	IF ((garPositionEndProcCalc[1] - T_Station_Parameter.T_StProcess.rPositionStartProc) <> 0.0) AND (T_Station_Parameter.T_OnlineChange.rWorkingSpeedForward <> 0.0) THEN
		T_Station_Work.THWWorkStation.TCtrlWork.iProgressBar_ZPos:=		REAL_TO_INT(100.0/(garPositionEndProcCalc[1] - T_Station_Parameter.T_StProcess.rPositionStartProc)
																			*(ptrTAxisZ^.T_LiveValue.lrActualPosition - T_Station_Parameter.T_StProcess.rPositionStartProc));
		T_Station_Work.THWWorkStation.TCtrlWork.iProgressBar_ZVel:=	REAL_TO_INT((100.0/T_Station_Parameter.T_OnlineChange.rWorkingSpeedForward)*ptrTAxisZ^.T_LiveValue.lrActualVelocity);
	ELSE
		T_Station_Work.THWWorkStation.TCtrlWork.iProgressBar_ZPos:=	0;
		T_Station_Work.THWWorkStation.TCtrlWork.iProgressBar_ZVel:=	0;
	END_IF;
	IF (T_Station_Work.THWWorkStation.TCtrlWork.iProgressBar_ZPos < 0) THEN
		T_Station_Work.THWWorkStation.TCtrlWork.iProgressBar_ZPos:=0;
	END_IF;
	IF (T_Station_Work.THWWorkStation.TCtrlWork.iProgressBar_ZVel < 0) THEN
		T_Station_Work.THWWorkStation.TCtrlWork.iProgressBar_ZVel:=0;
	END_IF;
(***************************************************************************************************************************************************)
(* Drehmoment Min-Max Werte oberhalb eines HC *)
rActTorque:=T_Station_Work.THWWorkStation.TCtrlWork.iProgressBar_Torque;
IF xStartFunction AND (iStationFunctionNr = 5) THEN
	IF (iStFct_StepPrc = 3) OR (iStFct_StepPrc = 4) THEN
		IF (rActTorque >= rTorqueMax) THEN
			rTorqueMax:=rActTorque;
		END_IF;
		IF (rActTorque >= rTorqueMin) THEN
			rTorqueMin:=rActTorque;
		END_IF;
	ELSE
		IF (T_Station_Work.THWWorkStation.TCtrlWork.iOverLimitCounterTorque >= 1) THEN
			IF (rTorqueMin <= rTorqueMin_Min) AND (rTorqueMin <> 0.0) AND (rTorqueMin >= 100.0)THEN
				rTorqueMin_Min:=rTorqueMin;
			END_IF;
			rTorqueMin:=0.0;
			IF (rTorqueMin_Min <> 99999.0) THEN
				T_Station_Work.THWWorkStation.TCtrlWork.rTorqueAfterHC_Min:=rTorqueMin_Min;
			END_IF;
		END_IF;
	END_IF;
	IF (rTorqueMax >= rTorqueMax_Max) THEN
		rTorqueMax_Max:=rTorqueMax;
	END_IF;
	T_Station_Work.THWWorkStation.TCtrlWork.rTorqueAfterHC_Max:=rTorqueMax_Max;
	IF (T_Station_Work.THWWorkStation.TCtrlWork.rTorqueAfterHC_Min <> 0.0) AND (T_Station_Work.THWWorkStation.TCtrlWork.rTorqueAfterHC_Min < 100.0) THEN
		T_Station_Work.THWWorkStation.TCtrlWork.rTorqueAfterHC_Min:=100.0;
	END_IF;
ELSE
	rTorqueMin:=0;
	rTorqueMax:=rActTorque;
	rTorqueMax_Max:=0;
	rTorqueMin_Min:=99999.0;
END_IF;
IF (T_Station_Work.THWWorkStation.TCtrlWork.rTorqueAfterHC_Min >= T_Station_Parameter.T_StProcess.iMaxTorque) THEN
	T_Station_Work.THWWorkStation.TCtrlWork.xTorqueAfterHC_Min_Overlimit:=TRUE;
ELSE
	T_Station_Work.THWWorkStation.TCtrlWork.xTorqueAfterHC_Min_Overlimit:=FALSE;
END_IF;
IF (T_Station_Work.THWWorkStation.TCtrlWork.rTorqueAfterHC_Max >= T_Station_Parameter.T_StProcess.iMaxTorque) THEN
	T_Station_Work.THWWorkStation.TCtrlWork.xTorqueAfterHC_Max_Overlimit:=TRUE;
ELSE
	T_Station_Work.THWWorkStation.TCtrlWork.xTorqueAfterHC_Max_Overlimit:=FALSE;
END_IF;
(***************************************************************************************************************************************************)
(* Ausgabe des Cursor für Progressbalken der Z Position für HC *)
IF xStartFunction AND (iStationFunctionNr = 5) AND (iStFct_StepPrc = 3) THEN
	IF T_Station_Work.THWWorkStation.TCtrlWork.xTorqueLastHC THEN
		IF (garPositionEndProcCalc[1] <> 0.0) THEN
			T_Station_Work.THWWorkStation.TCtrlWork.iHCTorquePos:=	REAL_TO_INT(100.0/(garPositionEndProcCalc[1] - T_Station_Parameter.T_StProcess.rPositionStartProc) *
																		(rStFct_SetZHCPosition - T_Station_Parameter.T_StProcess.rPositionStartProc) * 3.2);
		ELSE
			T_Station_Work.THWWorkStation.TCtrlWork.iHCTorquePos:=	0;
		END_IF;
	END_IF;
	IF T_Station_Work.THWWorkStation.TCtrlWork.xDeflectionLastHC THEN
		IF (garPositionEndProcCalc[1] <> 0.0) THEN
			T_Station_Work.THWWorkStation.TCtrlWork.iHCDeflectionPos:=	REAL_TO_INT(100.0/(garPositionEndProcCalc[1] - T_Station_Parameter.T_StProcess.rPositionStartProc) *
																			(rStFct_SetZHCPosition - T_Station_Parameter.T_StProcess.rPositionStartProc) * 3.2);
		ELSE
			T_Station_Work.THWWorkStation.TCtrlWork.iHCDeflectionPos:=0;
		END_IF;
	END_IF;
END_IF;
(***************************************************************************************************************************************************)
(* Auffangen HC beim ausfunken *)
IF xStartFunction AND (iStationFunctionNr = 5) AND (iStFct_StepPrc = 9) AND ptrTAxisZ^.T_CtrleSingle.xMovingForward THEN
	IF ptrTCylToolDeflection^.T_CtrleCyl.xStatePosOn THEN
		T_Station_Work.THWWorkStation.TCtrlWork.xHCSparkOut:=TRUE;
	END_IF;
END_IF;
(***************************************************************************************************************************************************)
END_FUNCTION_BLOCK
ACTION CtrlDCMotors:
(******************************************************************************************************************************************)
(* DC Motoren starten *)
(******************************************************************************************************************************************)
IF gxSuspensionONOFF AND (T_Station_Parameter.T_StProcess.rSuspensionBubblerSpeed <> 0) AND (gT_SafetyStatus.xEnergyONNormalMode OR gT_SafetyStatus.xEnergyONSetupModeASt1) THEN
	IF NOT(ptrTAxisBubbler^.T_CtrleDCAxis.xExecute) AND ptrTAxisBubbler^.T_CtrleDCAxis.xDone THEN
		IF NOT(ptrTAxisBubbler^.T_CtrleDCAxis.xReady) THEN
			ptrTAxisBubbler^.T_CtrleDCAxis.iFunction:=1;
			ptrTAxisBubbler^.T_CtrleDCAxis.xExecute:=TRUE;
		ELSIF NOT(ptrTAxisBubbler^.T_CtrleDCAxis.xPower) THEN
			ptrTAxisBubbler^.T_CtrleDCAxis.iFunction:=3;
			ptrTAxisBubbler^.T_CtrleDCAxis.xExecute:=TRUE;
		ELSIF ptrTAxisBubbler^.T_CtrleDCAxis.xNotMoving THEN
			ptrTAxisBubbler^.T_CtrleDCAxis.iFunction:=6;
			ptrTAxisBubbler^.T_CtrleDCAxis.lrVelocity:=T_Station_Parameter.T_StProcess.rSuspensionBubblerSpeed;				(* max 400.0 *)
			ptrTAxisBubbler^.T_CtrleDCAxis.tAcceleration:=T#0s;
			(*ptrTAxisBubbler^.T_CtrleDCAxis.tAcceleration:=T#500ms;
			ptrTAxisBubbler^.T_CtrleDCAxis.tDeceleration:=T#500ms;*)
			ptrTAxisBubbler^.T_CtrleDCAxis.xExecute:=TRUE;
		END_IF
	END_IF
ELSE
	IF NOT(ptrTAxisBubbler^.T_CtrleDCAxis.xExecute) AND ptrTAxisBubbler^.T_CtrleDCAxis.xDone THEN
		IF NOT(ptrTAxisBubbler^.T_CtrleDCAxis.xReady) THEN
			ptrTAxisBubbler^.T_CtrleDCAxis.iFunction:=1;
			ptrTAxisBubbler^.T_CtrleDCAxis.xExecute:=TRUE;
		ELSIF NOT(ptrTAxisBubbler^.T_CtrleDCAxis.xNotMoving) THEN
			ptrTAxisBubbler^.T_CtrleDCAxis.iFunction:=5;
			ptrTAxisBubbler^.T_CtrleDCAxis.xExecute:=TRUE;
		ELSIF ptrTAxisBubbler^.T_CtrleDCAxis.xPower THEN
			ptrTAxisBubbler^.T_CtrleDCAxis.iFunction:=4;
			ptrTAxisBubbler^.T_CtrleDCAxis.xExecute:=TRUE;
		END_IF
	END_IF
END_IF


IF gxSuspensionONOFF AND (T_Station_Parameter.T_StProcess.rSuspensionFeederSpeed <> 0) AND (gT_SafetyStatus.xEnergyONNormalMode OR gT_SafetyStatus.xEnergyONSetupModeASt1) THEN
	IF NOT(ptrTAxisFeedPump^.T_CtrleDCAxis.xExecute) AND ptrTAxisFeedPump^.T_CtrleDCAxis.xDone THEN
		IF NOT(ptrTAxisFeedPump^.T_CtrleDCAxis.xReady) THEN
			ptrTAxisFeedPump^.T_CtrleDCAxis.iFunction:=1;
			ptrTAxisFeedPump^.T_CtrleDCAxis.xExecute:=TRUE;
		ELSIF NOT(ptrTAxisFeedPump^.T_CtrleDCAxis.xPower) THEN
			ptrTAxisFeedPump^.T_CtrleDCAxis.iFunction:=3;
			ptrTAxisFeedPump^.T_CtrleDCAxis.xExecute:=TRUE;
		ELSIF NOT(IxSuspenstionFilled) AND NOT(ptrTAxisFeedPump^.T_CtrleDCAxis.xNotMoving) THEN
			ptrTAxisFeedPump^.T_CtrleDCAxis.iFunction:=5;
			ptrTAxisFeedPump^.T_CtrleDCAxis.xExecute:=TRUE;
		ELSIF ptrTAxisFeedPump^.T_CtrleDCAxis.xNotMoving THEN
			ptrTAxisFeedPump^.T_CtrleDCAxis.iFunction:=6;
			ptrTAxisFeedPump^.T_CtrleDCAxis.lrVelocity:=T_Station_Parameter.T_StProcess.rSuspensionFeederSpeed;			(* max 90.0 *)
			ptrTAxisFeedPump^.T_CtrleDCAxis.tAcceleration:=T#0s;
			(*ptrTAxisFeedPump^.T_CtrleDCAxis.tAcceleration:=T#500ms;
			ptrTAxisFeedPump^.T_CtrleDCAxis.tDeceleration:=T#500ms;*)
			ptrTAxisFeedPump^.T_CtrleDCAxis.xExecute:=TRUE;
		END_IF
	END_IF
ELSE
	IF NOT(ptrTAxisFeedPump^.T_CtrleDCAxis.xExecute) AND ptrTAxisFeedPump^.T_CtrleDCAxis.xDone THEN
		IF NOT(ptrTAxisFeedPump^.T_CtrleDCAxis.xNotMoving) THEN
			(*ptrTAxisFeedPump^.T_CtrleDCAxis.iFunction:=5;		funktioniert leider nicht, also über reset un iFunction:=1
			ptrTAxisFeedPump^.T_CtrleDCAxis.xExecute:=TRUE;*)
			ptrTAxisFeedPump^.T_CtrleDCAxis.xReset:=TRUE;
		ELSIF ptrTAxisFeedPump^.T_CtrleDCAxis.xPower THEN
			ptrTAxisFeedPump^.T_CtrleDCAxis.iFunction:=4;
			ptrTAxisFeedPump^.T_CtrleDCAxis.xExecute:=TRUE;
		ELSIF NOT(ptrTAxisFeedPump^.T_CtrleDCAxis.xReady) THEN
			ptrTAxisFeedPump^.T_CtrleDCAxis.iFunction:=1;
			ptrTAxisFeedPump^.T_CtrleDCAxis.xExecute:=TRUE;
		END_IF
	END_IF
END_IF
END_ACTION
ACTION CtrlDisableStation:
fbFTrig(CLK:=T_Station_Work.TControl.xEnable);
IF fbFTrig.Q THEN
	xInitSetEnable:=FALSE;
	xInitDelEnable:=FALSE;
	xRdyDisableStation:=FALSE;
END_IF;
IF (fbFTrig.Q OR xInitDelEnable) THEN
	IF NOT(xInitDelEnable) OR fbFTrig.Q THEN
		xReadyChkError:=FALSE;
		T_Station_Work.TControl.xDone:=FALSE;
		T_Station_Work.TControl.xError:=FALSE;
		xInitDelEnable:=TRUE;
		T_Station_Work.TControl.xRdy:=FALSE;
		iStepEnable:=100;
		iStationFunctionNr:=1;
		xInitStep:=FALSE;
	END_IF;
	CASE iStepEnable OF
		100:	IF NOT(xInitStep) THEN
				xInitStep:=TRUE;
				xStartFunction:=TRUE;
				xStFct_Reset:=TRUE;
			END_IF;
			IF NOT(xStFct_Reset) AND xStFct_End THEN
				(* Alle Funktionen Resetten *)
				IF (iStationFunctionNr < iMaxFunctionNr) THEN
					iStationFunctionNr:=iStationFunctionNr + 1;
					xStFct_Reset:=TRUE;
				ELSE
					xInitStep:=FALSE;
					xStartFunction:=FALSE;
					iStepEnable:=110;
				END_IF;
			(* Controlling für OnlineChange *)
				T_Station_Work.TCtrlOnlineChange.xLockChangeCylToolDeflectionForce:=TRUE;
				T_Station_Work.TCtrlOnlineChange.xLockChange_Z_WorkSpeedBackward:=TRUE;
				T_Station_Work.TCtrlOnlineChange.xLockChange_Z_WorkSpeedForward:=TRUE;
				T_Station_Work.TCtrlOnlineChange.xLockChange_S_WorkSpindleSpeed:=TRUE;
				T_Station_Work.TCtrlOnlineChange.xLockChangeCylToolTorqueLevel:=TRUE;
			END_IF;
		110:	IF NOT(xInitStep) THEN
				xInitStep:=TRUE;
				T_Station_Work.TControl.xResetHardware:=TRUE;
			END_IF;
			IF NOT(T_Station_Work.TControl.xResetHardware) THEN
				xInitStep:=FALSE;
				iStepEnable:=200;
			END_IF;
		200:	IF NOT(xInitStep) THEN
				xInitStep:=TRUE;
				IF T_Station_Work.TControl.xHardwareConfigError THEN
					T_Station_Work.TControl.xHardwareConfigError:=FALSE;
					T_Station_Work.TControl.xActiveHardware:=FALSE;
				ELSE
					xInitStep:=FALSE;
					iStepEnable:=300;
				END_IF;
				RETURN;
			END_IF;
			IF NOT(T_Station_Work.TControl.xError) OR xDontDeleteErrorFlag THEN
				T_Station_Work.TControl.xActiveHardware:=TRUE;
				xInitStep:=FALSE;
				iStepEnable:=300;
				RETURN;
			END_IF;
		300:	IF NOT(xInitStep) THEN	(* Alle Hardware Bausteine resetten *)
				xInitStep:=TRUE;
				ptrTAxisZ^.T_CtrleSingle.xReset:=TRUE;
				ptrTAxisS^.T_CtrleSingle.xReset:=TRUE;
				ptrTAxisBubbler^.T_CtrleDCAxis.xReset:=TRUE;
				ptrTAxisFeedPump^.T_CtrleDCAxis.xReset:=TRUE;
			END_IF;
			IF xTmp THEN
				RETURN;	(* Wait until all Drives finished *)
			END_IF;
			IF (NOT(ptrTAxisZ^.T_CtrleSingle.xReset) AND ptrTAxisZ^.T_CtrleSingle.xErr)
			OR (NOT(ptrTAxisS^.T_CtrleSingle.xReset) AND ptrTAxisS^.T_CtrleSingle.xErr)
			OR (NOT(ptrTAxisBubbler^.T_CtrleDCAxis.xReset) AND ptrTAxisBubbler^.T_CtrleDCAxis.xErr)
			OR (NOT(ptrTAxisFeedPump^.T_CtrleDCAxis.xReset) AND ptrTAxisFeedPump^.T_CtrleDCAxis.xErr) THEN
				xInitStep:=FALSE;
				iStepEnable:=400;
			END_IF;
			IF NOT(ptrTAxisZ^.T_CtrleSingle.xReset) AND ptrTAxisZ^.T_CtrleSingle.xDone
			AND NOT(ptrTAxisS^.T_CtrleSingle.xReset) AND ptrTAxisS^.T_CtrleSingle.xDone
			AND NOT(ptrTAxisBubbler^.T_CtrleDCAxis.xReset) AND ptrTAxisBubbler^.T_CtrleDCAxis.xDone
			AND NOT(ptrTAxisFeedPump^.T_CtrleDCAxis.xReset) AND ptrTAxisFeedPump^.T_CtrleDCAxis.xDone THEN
				T_Station_Work.TControl.xActiveHardware:=FALSE;
				xInitStep:=FALSE;
				xInitDelEnable:=FALSE;
				xSetEnd:=TRUE;
				xRdyDisableStation:=TRUE;
				IF xDontDeleteErrorFlag THEN
					T_Station_Work.TControl.xError:=TRUE;
				END_IF;
			END_IF;
		400:	IF NOT(xInitStep) THEN
				xInitStep:=TRUE;
				ptrTAxisZ^.T_CtrleSingle.iFunction:=1;
				ptrTAxisZ^.T_CtrleSingle.xExecute:=ptrTAxisZ^.T_CtrleSingle.xErr;
				ptrTAxisS^.T_CtrleSingle.iFunction:=1;
				ptrTAxisS^.T_CtrleSingle.xExecute:=ptrTAxisS^.T_CtrleSingle.xErr;
			END_IF;
			IF xTmp THEN
				RETURN;	(* Wait until all Drives finished *)
			END_IF;
			IF (NOT(ptrTAxisZ^.T_CtrleSingle.xExecute) AND ptrTAxisZ^.T_CtrleSingle.xErr) OR
			    (NOT(ptrTAxisS^.T_CtrleSingle.xExecute) AND ptrTAxisS^.T_CtrleSingle.xErr) THEN
				xInitStep:=FALSE;
				iStepEnable:=500;
			END_IF;
			IF NOT(ptrTAxisZ^.T_CtrleSingle.xExecute) AND ptrTAxisZ^.T_CtrleSingle.xDone OR
			    NOT(ptrTAxisS^.T_CtrleSingle.xExecute) AND ptrTAxisS^.T_CtrleSingle.xDone THEN
				T_Station_Work.TControl.xActiveHardware:=FALSE;
				xInitStep:=FALSE;
				xInitDelEnable:=FALSE;
				xSetEnd:=TRUE;
				xRdyDisableStation:=TRUE;
				IF xDontDeleteErrorFlag THEN
					T_Station_Work.TControl.xError:=TRUE;
				END_IF;
			END_IF;
		500:	T_Station_Work.TControl.xActiveHardware:=FALSE;
			T_Station_Work.TControl.diErrorNr:=1000000 + 16#F220;	(* Fehler / Error während disable (Ausschalten) der Station  *)
			T_Station_Work.TControl.xError:=TRUE;
			xDontDeleteErrorFlag:=TRUE;
			xInitStep:=FALSE;
			xInitDelEnable:=FALSE;
			xSetEnd:=TRUE;
			xRdyDisableStation:=TRUE;
	END_CASE;
END_IF;
END_ACTION
ACTION CtrlEnableStation:
fbRTrig(CLK:=T_Station_Work.TControl.xEnable);
IF fbRTrig.Q THEN
	xInitSetEnable:=FALSE;
	xInitDelEnable:=FALSE;
END_IF;
TONTimeOutEnablePart(IN:=T_Station_Work.TControl.xEnable AND xInitSetEnable,PT:=T#60s);
TONCalcMinTimeEnable(IN:=TRUE,PT:=T#9999s);
IF TONTimeOutEnablePart.Q THEN
	T_Station_Work.TControl.xEnable:=FALSE;
END_IF;
IF (fbRTrig.Q OR xInitSetEnable) THEN
	IF NOT(fbRTrig.Q) AND xReadyChkError THEN
		IF xSetError OR ptrTAxisZ^.T_CtrleSingle.xErr THEN
			IF (xTmp) AND NOT(xSetError) THEN
				RETURN;	(* Wait until all Actuators are not working *)
			END_IF;
			IF xSetError THEN
				xSetError:=FALSE;
				T_Station_Work.TControl.diErrorNr:=1000000 + diErrorNumber;
			ELSE
				ptrTAxisZ^.T_CtrleSingle.xReset:=ptrTAxisZ^.T_CtrleSingle.xErr;
				ptrTAxisS^.T_CtrleSingle.xReset:=ptrTAxisS^.T_CtrleSingle.xErr;
				ptrTAxisBubbler^.T_CtrleDCAxis.xReset:=ptrTAxisBubbler^.T_CtrleDCAxis.xErr;
				ptrTAxisFeedPump^.T_CtrleDCAxis.xReset:=ptrTAxisFeedPump^.T_CtrleDCAxis.xErr;
				IF ptrTAxisZ^.T_CtrleSingle.xErr THEN T_Station_Work.TControl.diErrorNr:=20000000 + ptrTAxisZ^.T_CtrleSingle.udiErrorID; END_IF;
				IF ptrTAxisS^.T_CtrleSingle.xErr THEN T_Station_Work.TControl.diErrorNr:=24000000 + ptrTAxisS^.T_CtrleSingle.udiErrorID; END_IF;
				IF ptrTAxisBubbler^.T_CtrleDCAxis.xErr THEN T_Station_Work.TControl.diErrorNr:=7000000 + ptrTAxisBubbler^.T_CtrleDCAxis.udiErrorID; END_IF;
				IF ptrTAxisFeedPump^.T_CtrleDCAxis.xErr THEN T_Station_Work.TControl.diErrorNr:=8000000 + ptrTAxisFeedPump^.T_CtrleDCAxis.udiErrorID; END_IF;
			END_IF;
			T_Station_Work.TControl.xEnable:=FALSE;
			xDontDeleteErrorFlag:=TRUE;
			RETURN;
		END_IF;
	END_IF;
	IF NOT(xInitSetEnable) OR fbRTrig.Q THEN
		xSetEnd:=FALSE;
		xInitSetEnable:=TRUE;
		T_Station_Work.TControl.xRdy:=FALSE;
		T_Station_Work.TControl.xDone:=FALSE;
		T_Station_Work.TControl.xError:=FALSE;
		T_Station_Work.TControl.diErrorNr:=0;
		iStepEnable:=100;
		iStationFunctionNr:=1;
		xInitStep:=FALSE;
		TONCalcMinTimeEnable(IN:=FALSE);
		RETURN;
	END_IF;
	CASE iStepEnable OF
		100:	IF NOT(xRdyDisableStation) AND NOT(gxHardwareOFF) AND NOT(gxAxisOFF) THEN
				iStepEnable:=110;
				RETURN;
			END_IF;
			IF NOT(xInitStep) THEN
				xInitStep:=TRUE;
				xStartFunction:=TRUE;
				xStFct_Reset:=TRUE;
				(* Initialisierung der HW *)
				T_Station_Work.TControl.xActiveHardware:=TRUE;
			(* Controlling für OnlineChange *)
				T_Station_Work.TCtrlOnlineChange.xLockChangeCylToolDeflectionForce:=FALSE;
				T_Station_Work.TCtrlOnlineChange.xLockChange_Z_WorkSpeedBackward:=TRUE;
				T_Station_Work.TCtrlOnlineChange.xLockChange_Z_WorkSpeedForward:=TRUE;
				T_Station_Work.TCtrlOnlineChange.xLockChange_S_WorkSpindleSpeed:=TRUE;
				T_Station_Work.TCtrlOnlineChange.xLockChangeCylToolTorqueLevel:=FALSE;
			END_IF;
			IF NOT(xStFct_Reset) AND xStFct_End THEN
				(* Alle Funktionen Resetten *)
				IF (iStationFunctionNr < iMaxFunctionNr) THEN
					iStationFunctionNr:=iStationFunctionNr + 1;
					xStFct_Reset:=TRUE;
				ELSE
					xInitStep:=FALSE;
					xStartFunction:=FALSE;
					iStepEnable:=200;
				END_IF;
			END_IF;
		110:	IF NOT(xInitStep) THEN
				xInitStep:=TRUE;
				IF T_Station_Work.TControl.xHardwareConfigError THEN
					T_Station_Work.TControl.xHardwareConfigError:=FALSE;
					T_Station_Work.TControl.xActiveHardware:=FALSE;
				ELSE
					xRdyDisableStation:=TRUE;
					xInitStep:=FALSE;
					iStepEnable:=100;
				END_IF;
				RETURN;
			END_IF;
			IF NOT(T_Station_Work.TControl.xError) THEN
				T_Station_Work.TControl.xActiveHardware:=TRUE;
				xRdyDisableStation:=TRUE;
				xInitStep:=FALSE;
				iStepEnable:=100;
				RETURN;
			END_IF;
		200:	IF NOT(xInitStep) THEN
				xInitStep:=TRUE;
				ptrTCylToolDeflection^.T_CtrleCyl.xReset:=TRUE;
				ptrTCylToolTorqueHC^.T_CtrleCyl.xReset:=TRUE;
				ptrTCylToolTorqueOverload^.T_CtrleCyl.xReset:=TRUE;
				ptrTTorqueSensorMeasRange^.T_CtrleCyl.xReset:=TRUE;
				ptrTTorqueSensorControl^.T_CtrleCyl.xReset:=TRUE;
				ptrTCylWorkpieceClamp^.T_CtrleCyl.xReset:=TRUE;
				ptrTValveAirTable^.T_CtrleCyl.xReset:=TRUE;
				ptrTValveVacuumTable^.T_CtrleCyl.xReset:=TRUE;
				ptrTCylBrakeReleaseZAxis^.T_CtrleCyl.xReset:=TRUE;
				ptrTAxisZ^.T_CtrleSingle.xReset:=TRUE;
				ptrTAxisS^.T_CtrleSingle.xReset:=TRUE;
				ptrTAxisBubbler^.T_CtrleDCAxis.xReset:=TRUE;
				ptrTAxisFeedPump^.T_CtrleDCAxis.xReset:=TRUE;
			END_IF;
			IF NOT(ptrTCylToolDeflection^.T_CtrleCyl.xReset) AND NOT(ptrTCylToolTorqueHC^.T_CtrleCyl.xReset)
			AND NOT(ptrTCylToolTorqueOverload^.T_CtrleCyl.xReset) AND NOT(ptrTCylBrakeReleaseZAxis^.T_CtrleCyl.xReset)
			AND NOT(ptrTTorqueSensorMeasRange^.T_CtrleCyl.xReset) AND NOT(ptrTTorqueSensorControl^.T_CtrleCyl.xReset)
			AND NOT(ptrTCylWorkpieceClamp^.T_CtrleCyl.xReset) AND NOT(ptrTValveAirTable^.T_CtrleCyl.xReset)
			AND NOT(ptrTValveVacuumTable^.T_CtrleCyl.xReset)
			AND NOT(ptrTAxisZ^.T_CtrleSingle.xReset) AND ptrTAxisZ^.T_CtrleSingle.xDone
			AND NOT(ptrTAxisS^.T_CtrleSingle.xReset) AND ptrTAxisS^.T_CtrleSingle.xDone
			AND NOT(ptrTAxisBubbler^.T_CtrleDCAxis.xReset) AND ptrTAxisBubbler^.T_CtrleDCAxis.xDone
			AND NOT(ptrTAxisFeedPump^.T_CtrleDCAxis.xReset) AND ptrTAxisFeedPump^.T_CtrleDCAxis.xDone THEN
				xInitStep:=FALSE;
				IF NOT(gxHardwareOFF) AND NOT(gxAxisOFF) THEN
					iStepEnable:=299;
				ELSE
					iStepEnable:=1100;
				END_IF;
			END_IF;
		299:	IF NOT(xInitStep) THEN
				xInitStep:=TRUE;
				ptrTAxisZ^.T_CtrleSingle.iFunction:=27;	(* Resetten des AX5000 Servo *)
				ptrTAxisZ^.T_CtrleSingle.xExecute:=TRUE;
			END_IF;
			IF NOT(ptrTAxisZ^.T_CtrleSingle.xExecute) AND ptrTAxisZ^.T_CtrleSingle.xDone THEN
				xInitStep:=FALSE;
				iStepEnable:=300;
			END_IF;
		300:	IF NOT(xInitStep) THEN
				xInitStep:=TRUE;
				ptrTAxisZ^.T_CtrleSingle.iFunction:=1;
				ptrTAxisZ^.T_CtrleSingle.xExecute:=TRUE;
				ptrTAxisS^.T_CtrleSingle.iFunction:=1;
				ptrTAxisS^.T_CtrleSingle.xExecute:=TRUE;
				ptrTAxisBubbler^.T_CtrleDCAxis.iFunction:=1;		(* Reset Axis *)
				ptrTAxisBubbler^.T_CtrleDCAxis.xExecute:=TRUE;
				ptrTAxisFeedPump^.T_CtrleDCAxis.iFunction:=1;	(* Reset Axis *)
				ptrTAxisFeedPump^.T_CtrleDCAxis.xExecute:=TRUE;
				iCountCycle:=0;
			END_IF;
			iCountCycle:=iCountCycle + 1;
			IF (iCountCycle >= 50) THEN
				xReadyChkError:=TRUE;	(* 50 SPS Zyklen warten bis die Übewachung der HW Error freigeschaltet werden kann *)
			END_IF;
			IF xTmp THEN
				RETURN;	(* Wait until all Drives finished *)
			END_IF;
			IF NOT(ptrTAxisZ^.T_CtrleSingle.xExecute) AND ptrTAxisZ^.T_CtrleSingle.xDone
			AND NOT(ptrTAxisS^.T_CtrleSingle.xExecute) AND ptrTAxisS^.T_CtrleSingle.xDone
			AND NOT(ptrTAxisBubbler^.T_CtrleDCAxis.xExecute) AND ptrTAxisBubbler^.T_CtrleDCAxis.xDone
			AND NOT(ptrTAxisFeedPump^.T_CtrleDCAxis.xExecute) AND ptrTAxisFeedPump^.T_CtrleDCAxis.xDone THEN
				xReadyChkError:=TRUE;
				xInitStep:=FALSE;
				iStepEnable:=400;
			END_IF;
		400:	IF NOT(xInitStep) THEN	(* Read Axis Parameter File-->wird nicht mehr gebraucht *)
				xInitStep:=TRUE;
				ptrTAxisZ^.T_CtrleSingle.sDeviceName:='Beckhoff';
				ptrTAxisS^.T_CtrleSingle.sDeviceName:='Maxon';
				ptrTAxisBubbler^.T_CtrleDCAxis.iFunction:=2;			(* Read Axis File *)
				ptrTAxisBubbler^.T_CtrleDCAxis.xExecute:=TRUE;
				ptrTAxisFeedPump^.T_CtrleDCAxis.iFunction:=2;		(* Read Axis File *)
				ptrTAxisFeedPump^.T_CtrleDCAxis.xExecute:=TRUE;
			END_IF;
			IF NOT(ptrTAxisZ^.T_CtrleSingle.xExecute) AND ptrTAxisZ^.T_CtrleSingle.xDone
			AND NOT(ptrTAxisS^.T_CtrleSingle.xExecute) AND ptrTAxisS^.T_CtrleSingle.xDone
			AND NOT(ptrTAxisBubbler^.T_CtrleDCAxis.xExecute) AND ptrTAxisBubbler^.T_CtrleDCAxis.xDone
			AND NOT(ptrTAxisFeedPump^.T_CtrleDCAxis.xExecute) AND ptrTAxisFeedPump^.T_CtrleDCAxis.xDone THEN
				xInitStep:=FALSE;
				iStepEnable:=500;
			END_IF;
		500:	IF NOT(xInitStep) THEN	(* Send Axis Parameter File-->wird nicht mehr gebraucht *)
				xInitStep:=TRUE;
				IF ptrTAxisBubbler^.T_CtrleDCAxis.xErr OR NOT(ptrTAxisBubbler^.T_CtrleDCAxis.xDone) THEN
					ptrTAxisBubbler^.T_CtrleDCAxis.iFunction:=1;
					ptrTAxisBubbler^.T_CtrleDCAxis.xExecute:=TRUE;
				END_IF;
				IF ptrTAxisFeedPump^.T_CtrleDCAxis.xErr OR NOT(ptrTAxisFeedPump^.T_CtrleDCAxis.xDone) THEN
					ptrTAxisFeedPump^.T_CtrleDCAxis.iFunction:=1;
					ptrTAxisFeedPump^.T_CtrleDCAxis.xExecute:=TRUE;
				END_IF;
			END_IF;
			IF NOT(ptrTAxisBubbler^.T_CtrleDCAxis.xExecute) AND ptrTAxisBubbler^.T_CtrleDCAxis.xDone
			AND NOT(ptrTAxisFeedPump^.T_CtrleDCAxis.xExecute) AND ptrTAxisFeedPump^.T_CtrleDCAxis.xDone THEN
				xInitStep:=FALSE;
				iStepEnable:=600;
			END_IF;
		600:	IF NOT(xInitStep) THEN	(* Keine BoxId mehr *)
				xInitStep:=TRUE;
				ptrTAxisBubbler^.T_CtrleDCAxis.iFunction:=1;			(* Reset Axis *)
				ptrTAxisBubbler^.T_CtrleDCAxis.xExecute:=TRUE;
				ptrTAxisFeedPump^.T_CtrleDCAxis.iFunction:=1;		(* Reset Axis *)
				ptrTAxisFeedPump^.T_CtrleDCAxis.xExecute:=TRUE;
			END_IF;
			IF NOT(ptrTAxisBubbler^.T_CtrleDCAxis.xExecute) AND ptrTAxisBubbler^.T_CtrleDCAxis.xDone
			AND NOT(ptrTAxisFeedPump^.T_CtrleDCAxis.xExecute) AND ptrTAxisFeedPump^.T_CtrleDCAxis.xDone THEN
				xInitStep:=FALSE;
				iStepEnable:=700;
			END_IF
		700:	IF NOT(xInitStep) THEN	(* Keine Konfigurationsfehler mehr *)
				xInitStep:=TRUE;
			END_IF;
			xInitStep:=FALSE;
			iStepEnable:=800;
		800:	IF NOT(xInitStep) THEN
				xInitStep:=TRUE;
				IF xSafetyCircuitOn THEN
					ptrTAxisZ^.T_CtrleSingle.iFunction:=3;
					ptrTAxisZ^.T_CtrleSingle.xExecute:=TRUE;
				END_IF;
			END_IF;
			IF NOT(ptrTAxisZ^.T_CtrleSingle.xExecute) AND ptrTAxisZ^.T_CtrleSingle.xDone AND (ptrTAxisZ^.T_CtrleSingle.xPower OR NOT(xSafetyCircuitOn)) THEN
				iStepEnable:=900;
				xInitStep:=FALSE;
			END_IF;
		900:	IF NOT(xInitStep) THEN
				xInitStep:=TRUE;
				ptrTAxisZ^.T_CtrleSingle.iFunction:=1;
				ptrTAxisZ^.T_CtrleSingle.xExecute:=TRUE;
				ptrTAxisS^.T_CtrleSingle.iFunction:=1;
				ptrTAxisS^.T_CtrleSingle.xExecute:=TRUE;
				ptrTAxisBubbler^.T_CtrleDCAxis.iFunction:=21;			(* Axisparameter senden *)
				ptrTAxisBubbler^.T_CtrleDCAxis.xExecute:=TRUE;
				ptrTAxisFeedPump^.T_CtrleDCAxis.iFunction:=21;		(* Axisparameter senden *)
				ptrTAxisFeedPump^.T_CtrleDCAxis.xExecute:=TRUE;
			END_IF;
			IF xTmp THEN
				RETURN;	(* Wait until all Drives finished *)
			END_IF;
			IF NOT(ptrTAxisZ^.T_CtrleSingle.xExecute) AND ptrTAxisZ^.T_CtrleSingle.xDone
			AND NOT(ptrTAxisS^.T_CtrleSingle.xExecute) AND ptrTAxisS^.T_CtrleSingle.xDone
			AND NOT(ptrTAxisBubbler^.T_CtrleDCAxis.xExecute) AND ptrTAxisBubbler^.T_CtrleDCAxis.xDone
			AND NOT(ptrTAxisFeedPump^.T_CtrleDCAxis.xExecute) AND ptrTAxisFeedPump^.T_CtrleDCAxis.xDone THEN
				xInitStep:=FALSE;
				iStepEnable:=1000;
			END_IF;
		1000:IF NOT(xInitStep) THEN
				xInitStep:=TRUE;
				IF T_Station_Parameter.T_AxisState.xReferencedZAxis THEN
					IF NOT(xFirstBooting) THEN
						ptrTAxisZ^.T_CtrleSingle.rSetPosition:=	ptrTAxisZ^.T_LiveValue.lrActualPosition -
																T_Station_Parameter.T_AxisState.rPositionReferenceZAxis;
						ptrTAxisZ^.T_CtrleSingle.iFunction:=11;		(* Position setzen *)
						ptrTAxisZ^.T_CtrleSingle.xExecute:=TRUE;
					END_IF;
				END_IF;
				xFirstBooting:=TRUE;
			END_IF;
			IF NOT(ptrTAxisZ^.T_CtrleSingle.xExecute) AND ptrTAxisZ^.T_CtrleSingle.xDone THEN
				iStepEnable:=1100;
				xInitStep:=FALSE;
			END_IF;
		1100:IF NOT(xInitStep) THEN
				xInitStep:=TRUE;
				(* Zylinder für Auslenkung-->mit Workauslenkkraft *)
				ptrTCylToolDeflection^.T_CtrleCyl.iFunction:=2;
				ptrTCylToolDeflection^.T_Config.tDelayOn:=T#0.3s;
				ptrTCylToolDeflection^.T_CtrleCyl.T_Analog.rForceIn:=T_Station_Parameter.T_OnlineChange.rForceDeflection;
				ptrTCylToolDeflection^.T_CtrleCyl.xExecute:=TRUE;
				IF  (T_Station_Parameter.T_Fct_SpindleCalibration.arOffsetToolDeflection[1] <= 0.0) THEN
					T_Station_Parameter.T_Fct_SpindleCalibration.arOffsetToolDeflection[1]:=6.0;
				END_IF;
				IF  (T_Station_Parameter.T_Fct_SpindleCalibration.arOffsetToolTorque[1] <= 0.0) THEN
					T_Station_Parameter.T_Fct_SpindleCalibration.arOffsetToolTorque[1]:=6.0;
				END_IF;
			END_IF;
			IF NOT(ptrTCylToolDeflection^.T_CtrleCyl.xExecute) AND ptrTCylToolDeflection^.T_CtrleCyl.xDone THEN
				iStepEnable:=1101;
				xInitStep:=FALSE;
			END_IF;
		1101:IF (TONCalcMinTimeEnable.ET >= T#3.5s) THEN	(* Mindestens diese Zeit muss eingehalten werden, damit bei unterschidlichen Laufzeiten von Maschinen der Progressbalken beim auftsarten in etwa immer gleich dauert *)
				iStepEnable:=1200;
				xInitStep:=FALSE;
				xWaitAxisVoltageBooting:=FALSE;
			END_IF;
		1200:xReadyChkError:=FALSE;
			xInitStep:=FALSE;
			xInitSetEnable:=FALSE;
			T_Station_Work.TControl.xRdy:=TRUE;
			xSetEnd:=TRUE;
			xStFct_ForceStationError:=FALSE;
	END_CASE;
END_IF;
END_ACTION
ACTION CtrlErrorStation:
IF (xStationError OR xForceHWError OR xStFct_ForceStationError OR (xStFct_Error AND T_Station_Work.TControl.xRdy AND NOT(xSetEnd))) AND NOT(T_Station_Work.TControl.xSecurityCircuitOff) THEN
	IF NOT(xInitError) THEN
		IF xForceHWError THEN
			T_Station_Work.TControl.diErrorNr:=0;
			xForceHWError:=FALSE;
		END_IF;
		iSettledErrFromFunction:=iStationFunctionNr;
		xStationError:=TRUE;
		xTmpStationError:=TRUE;
		xInitError:=TRUE;
		xAxisErrorActive:=FALSE;
		T_Station_Work.TControl.diErrorNr:=0;
		xStFct_ForceStationError:=FALSE;
		IF ptrTAxisZ^.T_CtrleSingle.xErr THEN
			IF (T_Station_Work.TControl.diErrorNr = 0) THEN
				T_Station_Work.TControl.diErrorNr:=20000000 + ptrTAxisZ^.T_CtrleSingle.udiErrorID;
			END_IF;
			ptrTAxisZ^.T_CtrleSingle.xReset:=TRUE;
			xAxisErrorActive:=TRUE;
		END_IF;
		IF ptrTAxisS^.T_CtrleSingle.xErr THEN
			IF (T_Station_Work.TControl.diErrorNr = 0) THEN
				T_Station_Work.TControl.diErrorNr:=24000000 + ptrTAxisS^.T_CtrleSingle.udiErrorID;
			END_IF;
			ptrTAxisS^.T_CtrleSingle.xReset:=TRUE;
			xAxisErrorActive:=TRUE;
		END_IF;
		IF ptrTCylBrakeReleaseZAxis^.T_CtrleCyl.xErr THEN
			IF (T_Station_Work.TControl.diErrorNr = 0) THEN
				T_Station_Work.TControl.diErrorNr:=42000000 + ptrTCylBrakeReleaseZAxis^.T_CtrleCyl.udiErrorID;
			END_IF;
			ptrTCylBrakeReleaseZAxis^.T_CtrleCyl.xReset:=TRUE;
		END_IF;
		IF (T_Station_Work.TControl.diErrorNr = 0) THEN	(* General Error-->No Hardware Error  1000000 - 1999999*)
			T_Station_Work.TControl.diErrorNr:=1000000 + diStFct_ErrorNr;
		END_IF;
		xStFct_QuitErr:=NOT(xStFct_End) AND xStFct_Error;
		IF NOT(xStFct_QuitErr) AND NOT(xStFct_End) THEN
			xForceResetAxis:=TRUE;
			xStFct_Reset:=TRUE;
			xStFct_SetEnd:=TRUE;
			StationFunction_Ctrl_End;
		END_IF;
		TONWaitReset(IN:=FALSE);
	END_IF;
	xStFct_QuitErr:=NOT(xStFct_End) AND xStFct_Error;
	IF (xStFct_End OR xForceResetAxis) AND xTmpStationError THEN
		xStartFunction:=FALSE;
		TONWaitReset(IN:=TRUE,PT:=T#500ms);
		IF TONWaitReset.Q THEN
			xStepError:=FALSE;
			xTmpStationError:=FALSE;
			xReadyToQuitErr:=TRUE;
			T_Station_Work.TControl.xError:=TRUE;
			T_Station_Work.TControl.xDone:=FALSE;
			xForceResetAxis:=FALSE;
		END_IF;
	END_IF;
	IF T_Station_Work.TControl.xQuitError AND NOT(xStFct_QuitErr) AND xReadyToQuitErr THEN
		xInitError:=FALSE;
		T_Station_Work.TControl.xQuitError:=FALSE;
		xSetEnd:=TRUE;
	END_IF;
ELSE
	(* Gilt für Fehler die ausserhalb der Station gesetzt werden und diese zurücksetzen zu können *)
	IF T_Station_Work.TControl.xQuitError THEN
		T_Station_Work.TControl.xQuitError:=FALSE;
		xSetEnd:=TRUE;
	END_IF;
	(* Überwachung Drehmoment Überlast *)
	IF (iStationFunctionNr <> 4) AND (iStationFunctionNr <> 5) THEN
		IF ptrTCylToolTorqueOverload^.T_CtrleCyl.xStatePosOn OR ptrTSensorTorqueOverload^.T_CtrleCyl.xStatePosOn THEN
			IF NOT(ptrTAxisS^.T_CtrleSingle.xExecute) AND NOT(ptrTAxisS^.T_CtrleSingle.xNotMoving) AND ptrTAxisS^.T_CtrleSingle.xDone THEN
				ptrTAxisS^.T_CtrleSingle.iFunction:=5;
				ptrTAxisS^.T_CtrleSingle.xExecute:=TRUE;
				gxSpindleOverloadError:=TRUE;
			END_IF;
		END_IF;
	END_IF;
END_IF;
END_ACTION
ACTION CtrlMainStation:
IF T_Station_Work.TControl.xRdy THEN
	T_Station_Work.TControl.xReferenced:=T_Station_Parameter.T_AxisState.xReferencedZAxis;
END_IF;
IF (T_Station_Work.TControl.xExecute OR xTmpStart) AND T_Station_Work.TControl.xRdy AND NOT(xSetEnd) THEN
	IF NOT(xInitStart) THEN
		xInitStart:=TRUE;
		xTmpStart:=TRUE;
		T_Station_Work.TControl.xExecute:=FALSE;
		T_Station_Work.TControl.xDone:=FALSE;
		xStFct_Start:=TRUE;
		xStartFunction:=TRUE;
		iStationFunctionNr:=T_Station_Work.TControl.iFunctNr;
		T_Station_Work.TControl.xAbord:=FALSE;
		xStFct_HardwareError:=xStFct_ErrorActuator:=xStFct_InitError:=FALSE;
		xStFct_ForceSetSpeedZAxis:=FALSE;
		xStFct_ForceSetSpeedTorqueZAxis:=FALSE;
		T_Station_Work.THWWorkStation.TCtrlWork.xToolInfeeded:=FALSE;
		xMaxTorqueActive:=FALSE;
		xPartDiscNotInPosition:=FALSE;
	END_IF;
	IF T_Station_Work.TControl.xStop THEN
		IF NOT(xInitStop) THEN
			xInitStop:=TRUE;
			xStFct_Stop:=TRUE;
		END_IF;
		IF NOT(xStFct_Stop) THEN
			xInitStop:=FALSE;
			T_Station_Work.TControl.xStop:=FALSE;
			xTmpStopFunction:=TRUE;
		END_IF;
	END_IF;
	IF T_Station_Work.TControl.xExecute AND xTmpStopFunction AND NOT(xStFct_Abord) THEN
		T_Station_Work.TControl.xExecute:=FALSE;
		xTmpStopFunction:=FALSE;
		xStFct_Start:=TRUE;
	END_IF;
	IF T_Station_Work.TControl.xAbord AND xTmpStopFunction THEN
		T_Station_Work.TControl.xAbord:=FALSE;
		xTmpStopFunction:=FALSE;
		xStFct_Start:=FALSE;
		xStFct_Abord:=TRUE;
	END_IF;
	IF NOT(xStFct_Start) AND xStFct_End AND NOT(xStationError) THEN
		xTmpStart:=FALSE;
		xInitStart:=FALSE;
		xSetEnd:=TRUE;
	END_IF;
END_IF;
END_ACTION
ACTION CtrlSafetySwitch_ON_OFF:
TONCheckAxisVoltagBooting(IN:=xStartTimer,PT:=T#60s);
IF NOT(T_TwinSafeOut.QxContactorMasterModul400VCh1) OR NOT(T_TwinSafeOut.QxContactorMasterModul400VCh2) THEN
	xStartTimer:=TRUE;
ELSE
	xStartTimer:=FALSE;
END_IF;
IF TONCheckAxisVoltagBooting.Q THEN
	xWaitAxisVoltageBooting:=TRUE;
END_IF;
TONWaitCheckCylinder(IN:=TRUE,PT:=T#1s);
IF (T_Station_Work.TControl.xSecurityCircuitOn OR T_Station_Work.TControl.xSecurityCircuitOff OR xSecurityCircuitOn OR xSecurityCircuitOff) AND NOT(xInitSetEnable) AND NOT(xInitDelEnable) AND NOT(xStationError) THEN
	TONWaitCheckCylinder(IN:=FALSE);
	T_Station_Work.TControl.xBlockCheckZylinder:=TRUE;
	IF NOT(xSecurityCircuitOn) AND NOT(xSecurityCircuitOff) THEN
		xSecurityCircuitOn:=T_Station_Work.TControl.xSecurityCircuitOn;
		xSecurityCircuitOff:=T_Station_Work.TControl.xSecurityCircuitOff;
		iStepSecCircuit:=1;
		xInitSecCircuit:=FALSE;
		T_Station_Work.TControl.xDone:=FALSE;
		TONCheckError(IN:=FALSE);
	END_IF;
	IF xSecurityCircuitOn THEN
		IF T_Station_Work.TControl.xSecurityCircuitOff THEN
			T_Station_Work.TControl.xSecurityCircuitOn:=FALSE;
			xSecurityCircuitOn:=FALSE;
		END_IF;
	END_IF;
	IF xSecurityCircuitOff THEN
		IF T_Station_Work.TControl.xSecurityCircuitOn THEN
			T_Station_Work.TControl.xSecurityCircuitOff:=FALSE;
			xSecurityCircuitOff:=FALSE;
		END_IF;
	END_IF;
	CASE iStepSecCircuit OF
	1:	IF gxHardwareOFF OR gxAxisOFF THEN
			xInitSecCircuit:=FALSE;
			iStepSecCircuit:=60;
			RETURN;
		END_IF;
		IF xSecurityCircuitOff THEN
			TONCheckError(IN:=TRUE,PT:=T#50ms);
			IF TONCheckError.Q THEN
				TONCheckError(IN:=FALSE);
				iStepSecCircuit:=iStepSecCircuit + 1;
			END_IF;
		ELSE
			iStepSecCircuit:=iStepSecCircuit + 1;
		END_IF;
		ptrTAxisZ^.T_CtrleSingle.xReset:=TRUE;
		(* Controlling für OnlineChange *)
		IF xSecurityCircuitOn THEN
			T_Station_Work.TCtrlOnlineChange.xLockChangeCylToolDeflectionForce:=FALSE;
			T_Station_Work.TCtrlOnlineChange.xLockChange_Z_WorkSpeedBackward:=TRUE;
			T_Station_Work.TCtrlOnlineChange.xLockChange_Z_WorkSpeedForward:=TRUE;
			T_Station_Work.TCtrlOnlineChange.xLockChange_S_WorkSpindleSpeed:=TRUE;
			T_Station_Work.TCtrlOnlineChange.xLockChangeCylToolTorqueLevel:=FALSE;
		ELSE
			T_Station_Work.TCtrlOnlineChange.xLockChangeCylToolDeflectionForce:=TRUE;
			T_Station_Work.TCtrlOnlineChange.xLockChange_Z_WorkSpeedBackward:=TRUE;
			T_Station_Work.TCtrlOnlineChange.xLockChange_Z_WorkSpeedForward:=TRUE;
			T_Station_Work.TCtrlOnlineChange.xLockChange_S_WorkSpindleSpeed:=TRUE;
			T_Station_Work.TCtrlOnlineChange.xLockChangeCylToolTorqueLevel:=TRUE;
		END_IF;
	2:	T_Station_Work.TControl.xRdy:=FALSE;
		IF NOT(xInitSecCircuit) THEN
			xInitSecCircuit:=TRUE;
			xStFct_Reset:=TRUE;
			iStationFunctionNr:=1;
			xStartFunction:=TRUE;
		END_IF;
		IF NOT(xStFct_Reset) AND xStFct_End THEN
			(* Alle Funktionen Resetten *)
			xInitSecCircuit:=FALSE;
			iStepSecCircuit:=10;
			xStartFunction:=FALSE;
		END_IF;
	10:	IF NOT(xInitSecCircuit) THEN
			xInitSecCircuit:=TRUE;
			T_Station_Work.TControl.xResetHardware:=TRUE;
			ptrTAxisBubbler^.T_CtrleDCAxis.xReset:=TRUE;
			ptrTAxisFeedPump^.T_CtrleDCAxis.xReset:=TRUE;
		END_IF;
		IF NOT(T_Station_Work.TControl.xResetHardware)
		AND NOT(ptrTAxisBubbler^.T_CtrleDCAxis.xReset) AND NOT(ptrTAxisFeedPump^.T_CtrleDCAxis.xReset) THEN
			xInitSecCircuit:=FALSE;
			iStepSecCircuit:=20;
		END_IF;
	20:	IF NOT(xInitSecCircuit) THEN
			xInitSecCircuit:=TRUE;
			ptrTAxisBubbler^.T_CtrleDCAxis.iFunction:=1;					(* Reset Axis *)
			ptrTAxisBubbler^.T_CtrleDCAxis.xExecute:=TRUE;
			ptrTAxisFeedPump^.T_CtrleDCAxis.iFunction:=1;					(* Reset Axis *)
			ptrTAxisFeedPump^.T_CtrleDCAxis.xExecute:=TRUE;
		END_IF;
		IF (NOT(ptrTAxisBubbler^.T_CtrleDCAxis.xExecute) AND (ptrTAxisBubbler^.T_CtrleDCAxis.xDone OR ptrTAxisBubbler^.T_CtrleDCAxis.xErr))
		AND (NOT(ptrTAxisFeedPump^.T_CtrleDCAxis.xExecute) AND (ptrTAxisFeedPump^.T_CtrleDCAxis.xDone OR ptrTAxisFeedPump^.T_CtrleDCAxis.xErr)) THEN
			xInitSecCircuit:=FALSE;
			iStepSecCircuit:=30;
		END_IF;
	30:	IF NOT(xInitSecCircuit) THEN
			xInitSecCircuit:=TRUE;
			ptrTAxisZ^.T_CtrleSingle.iFunction:=4;
			ptrTAxisZ^.T_CtrleSingle.xExecute:=TRUE;
			ptrTAxisS^.T_CtrleSingle.iFunction:=4;
			ptrTAxisS^.T_CtrleSingle.xExecute:=TRUE;
		END_IF;
		IF (NOT(ptrTAxisZ^.T_CtrleSingle.xExecute) AND (ptrTAxisZ^.T_CtrleSingle.xDone OR ptrTAxisZ^.T_CtrleSingle.xErr)) AND
		    (NOT(ptrTAxisS^.T_CtrleSingle.xExecute) AND (ptrTAxisS^.T_CtrleSingle.xDone OR ptrTAxisS^.T_CtrleSingle.xErr)) THEN
			IF ptrTAxisZ^.T_CtrleSingle.xErr THEN
				xInitSecCircuit:=FALSE;
				iStepSecCircuit:=10;
			ELSE
				xInitSecCircuit:=FALSE;
				iStepSecCircuit:=40;
			END_IF;
		END_IF;
	40:	IF NOT(xInitSecCircuit) THEN
			xInitSecCircuit:=TRUE;
			(* Resetten der Aktuatoren *)
			ptrTCylToolDeflection^.T_CtrleCyl.xReset:=TRUE;
			ptrTCylBrakeReleaseZAxis^.T_CtrleCyl.xReset:=TRUE;
			ptrTCylToolTorqueHC^.T_CtrleCyl.xReset:=TRUE;
			ptrTCylToolTorqueOverload^.T_CtrleCyl.xReset:=TRUE;

(*			ptrTCylWorkpieceClamp^.T_CtrleCyl.xReset:=TRUE;
			ptrTValveAirTable^.T_CtrleCyl.xReset:=TRUE;
			ptrTValveVacuumTable^.T_CtrleCyl.xReset:=TRUE;*)
		END_IF;
		IF NOT(ptrTCylToolDeflection^.T_CtrleCyl.xReset) AND NOT(ptrTCylToolTorqueHC^.T_CtrleCyl.xReset) AND
		     NOT(ptrTCylToolTorqueOverload^.T_CtrleCyl.xReset) AND NOT(ptrTCylBrakeReleaseZAxis^.T_CtrleCyl.xReset) AND
		     NOT(ptrTCylWorkpieceClamp^.T_CtrleCyl.xReset) AND NOT(ptrTValveAirTable^.T_CtrleCyl.xReset) AND
		     NOT(ptrTValveVacuumTable^.T_CtrleCyl.xReset) THEN
			xInitSecCircuit:=FALSE;
			IF xWaitAxisVoltageBooting AND (xSafetyCircuitOn) THEN
				iStepSecCircuit:=45;
			ELSE
				iStepSecCircuit:=50;
			END_IF;
		END_IF;
	45:	IF NOT(xInitSecCircuit) THEN
			xInitSecCircuit:=TRUE;
			TONWaitAxisCurrentSwitchON(IN:=FALSE);
		END_IF;
		TONWaitAxisCurrentSwitchON(IN:=TRUE,PT:=T#2s);
		IF TONWaitAxisCurrentSwitchON.Q THEN	(* Warten bis Zwischenkreisspannung aufgebaut ist, da es mehr als 1 Minute ausgeschaltet war *)
			xWaitAxisVoltageBooting:=FALSE;
			xInitSecCircuit:=FALSE;
			iStepSecCircuit:=50;
		END_IF;
	50:	IF NOT(xInitSecCircuit) THEN
			xInitSecCircuit:=TRUE;
			IF xSafetyCircuitOn THEN
				ptrTAxisZ^.T_CtrleSingle.iFunction:=3;
				ptrTAxisZ^.T_CtrleSingle.xExecute:=TRUE;
				ptrTCylToolDeflection^.T_CtrleCyl.iFunction:=2;
				ptrTCylToolDeflection^.T_CtrleCyl.T_Analog.rForceIn:=T_Station_Parameter.T_OnlineChange.rForceDeflection;
				ptrTCylToolDeflection^.T_CtrleCyl.xExecute:=TRUE;
				ptrTCylToolTorqueHC^.T_CtrleCyl.iFunction:=2;
				ptrTCylToolTorqueHC^.T_CtrleCyl.T_Analog.rForceIn:=T_Station_Parameter.T_OnlineChange.rTorqueLevelHC;
				ptrTCylToolTorqueHC^.T_CtrleCyl.xExecute:=TRUE;
				ptrTCylToolTorqueOverload^.T_CtrleCyl.iFunction:=2;
				ptrTCylToolTorqueOverload^.T_CtrleCyl.T_Analog.rForceIn:=T_Station_Parameter.T_StProcess.rTorqueLevel_Overload;
				ptrTCylToolTorqueOverload^.T_CtrleCyl.xExecute:=TRUE;
				ptrTCylBrakeReleaseZAxis^.T_CtrleCyl.iFunction:=1;
				ptrTCylBrakeReleaseZAxis^.T_CtrleCyl.xExecute:=TRUE;
(*				ptrTCylWorkpieceClamp^.T_CtrleCyl.iFunction:=1;
				ptrTCylWorkpieceClamp^.T_CtrleCyl.xExecute:=TRUE;
				ptrTValveAirTable^.T_CtrleCyl.iFunction:=1;
				ptrTValveAirTable^.T_CtrleCyl.xExecute:=TRUE;
				ptrTValveVacuumTable^.T_CtrleCyl.iFunction:=1;
				ptrTValveVacuumTable^.T_CtrleCyl.xExecute:=TRUE;*)
			END_IF;
		END_IF;
		IF NOT(ptrTAxisZ^.T_CtrleSingle.xExecute) AND ptrTAxisZ^.T_CtrleSingle.xDone THEN
			xInitSecCircuit:=FALSE;
			iStepSecCircuit:=60;
			IF  (T_Station_Parameter.T_Fct_SpindleCalibration.arOffsetToolDeflection[1] <= 0.0) THEN
				T_Station_Parameter.T_Fct_SpindleCalibration.arOffsetToolDeflection[1]:=6.0;
			END_IF;
			IF (T_Station_Parameter.T_Fct_SpindleCalibration.arOffsetToolTorque[1] <= 0.0) THEN
				T_Station_Parameter.T_Fct_SpindleCalibration.arOffsetToolTorque[1]:=3.0;
			END_IF;
		END_IF;
	60:	T_Station_Work.TControl.xRdy:=TRUE;
		T_Station_Work.TControl.xSecurityCircuitOn:=FALSE;
		T_Station_Work.TControl.xSecurityCircuitOff:=FALSE;
		xSecurityCircuitOn:=FALSE;
		xSecurityCircuitOff:=FALSE;
		iStepSecCircuit:=1;
		xInitSecCircuit:=FALSE;
		xSetEnd:=TRUE;
		xStFct_ForceStationError:=FALSE;
	END_CASE;
ELSE
	T_Station_Work.TControl.xSecurityCircuitOn:=FALSE;
	T_Station_Work.TControl.xSecurityCircuitOff:=FALSE;
	xSecurityCircuitOn:=FALSE;
	xSecurityCircuitOff:=FALSE;
	iStepSecCircuit:=1;
	xInitSecCircuit:=FALSE;
	TONCheckError(IN:=FALSE);
	IF TONWaitCheckCylinder.Q THEN
		T_Station_Work.TControl.xBlockCheckZylinder:=FALSE;
		IF ptrTAxisBubbler^.T_CtrleDCAxis.xErr THEN
			ptrTAxisBubbler^.T_CtrleDCAxis.iFunction:=1;
			ptrTAxisBubbler^.T_CtrleDCAxis.xExecute:=TRUE;
		END_IF;
		IF ptrTAxisFeedPump^.T_CtrleDCAxis.xErr THEN
			ptrTAxisFeedPump^.T_CtrleDCAxis.iFunction:=1;
			ptrTAxisFeedPump^.T_CtrleDCAxis.xExecute:=TRUE;
		END_IF;
	END_IF;
END_IF;
END_ACTION
ACTION StationFunction_CheckOverload:
(* Überwachung Drehmoment Überlast *)
IF gxHardwareOFF THEN
	RETURN;
END_IF;
CASE T_ExchgParam.bToolSpindleActive OF
1:	(* Maxon Spindel *)
	IF ptrTCylToolTorqueOverload^.T_CtrleCyl.xStatePosOn THEN
		xStFct_Overload_StopProcess:=TRUE;
	END_IF;
	IF xStFct_Overload_StopProcess THEN
		CASE iStFct_Overload_StopProcess OF
		1:	T_Station_Work.TCtrlOnlineChange.xLockChange_Z_WorkSpeedForward:=TRUE;
			T_Station_Work.TCtrlOnlineChange.xLockChange_Z_WorkSpeedBackward:=TRUE;
			T_Station_Work.TCtrlOnlineChange.xLockChange_S_WorkSpindleSpeed:=TRUE;
			IF (NOT(ptrTAxisZ^.T_CtrleSingle.xNotMoving) OR NOT(ptrTAxisZ^.T_CtrleSingle.xDone)) AND
	     		    NOT((ptrTAxisZ^.T_CtrleSingle.iFunction = 5) AND NOT(ptrTAxisZ^.T_CtrleSingle.xDone)) THEN
				ptrTAxisZ^.T_CtrleSingle.iFunction:=5;
				ptrTAxisZ^.T_CtrleSingle.xExecute:=TRUE;
				iStFct_Overload_StopProcess:=iStFct_Overload_StopProcess + 1;
			ELSE
				iStFct_Overload_StopProcess:=iStFct_Overload_StopProcess + 1;
			END_IF;
			IF NOT(ptrTAxisS^.T_CtrleSingle.xExecute) AND NOT(ptrTAxisS^.T_CtrleSingle.xNotMoving) THEN
				ptrTAxisS^.T_CtrleSingle.iFunction:=5;
				ptrTAxisS^.T_CtrleSingle.xExecute:=TRUE;
			END_IF;
			RETURN;
		2:	IF NOT(ptrTAxisZ^.T_CtrleSingle.xExecute) AND ptrTAxisZ^.T_CtrleSingle.xDone AND
			    NOT(ptrTAxisS^.T_CtrleSingle.xExecute) AND ptrTAxisS^.T_CtrleSingle.xDone THEN
				T_Station_Work.THWWorkStation.TCtrlWork.xWorkingFinished:=TRUE;
				T_Station_Work.THWWorkStation.TCtrlWork.bPartQuality:=8;(* < Bearb. abgbr. > *)
				xStFct_HardwareError:=TRUE;
				diStFct_TmpErrorNr:=15;		(* Wz Drehmoment Überlast Aktiv *)
			END_IF;
			RETURN;
		END_CASE;
	END_IF;
2,3:	(* Beckhoff Spindel *)
	IF (T_Station_Parameter.T_StProcess.iWorkControlType <= 1) THEN
		IF (T_Station_Parameter.T_OnlineChange.rTorqueLevelHC <> 0.0) THEN
			CASE T_ExchgParam.bToolSpindleActive OF
			2:	(* Beckhoff Spindel L *)
				rTorquePercent:=REAL_TO_INT(100.0/T_Station_Parameter.T_OnlineChange.rTorqueLevelHC*T_Station_Parameter.T_TorqueSystem_L.rActual_Torque);
			3:	(* Beckhoff Spindel M *)
				rTorquePercent:=REAL_TO_INT(100.0/T_Station_Parameter.T_OnlineChange.rTorqueLevelHC*T_Station_Parameter.T_TorqueSystem_M.rActual_Torque);
			END_CASE;
		END_IF;
	END_IF;

	IF (T_Station_Parameter.T_StProcess.iWorkControlType = 2) THEN
		IF (T_Station_Parameter.T_StProcess.rZ_PID_Torque <> 0.0) THEN
			rTorquePercent:=REAL_TO_INT(100.0/T_Station_Parameter.T_StProcess.rZ_PID_Torque*rTorqueSpindleSensor);
		END_IF;
	END_IF

	IF (T_Station_Parameter.T_StProcess.iWorkControlType = 3) THEN
		IF (T_Station_Parameter.T_OnlineChange.rTorqueLevelHC <> 0.0) THEN
			rTorquePercent:=REAL_TO_INT(100.0/T_Station_Parameter.T_OnlineChange.rTorqueLevelHC*rTorqueSpindleSensor);
		END_IF;
	END_IF;

	IF (rTorquePercent >= T_Station_Parameter.T_StProcess.iMaxTorque) THEN
		IF (rTorqueMax < T_Station_Parameter.T_StProcess.iMaxTorque) THEN
			rTorqueMax:=T_Station_Parameter.T_StProcess.iMaxTorque;
		END_IF;
		xMaxTorqueActive:=TRUE;
	END_IF;

	IF ptrTSensorTorqueOverload^.T_CtrleCyl.xStatePosOn OR xMaxTorqueActive THEN
		xStFct_Overload_StopProcess:=TRUE;
	END_IF;
	IF xStFct_Overload_StopProcess THEN
		CASE iStFct_Overload_StopProcess OF
		1:	T_Station_Work.TCtrlOnlineChange.xLockChange_Z_WorkSpeedForward:=TRUE;
			T_Station_Work.TCtrlOnlineChange.xLockChange_Z_WorkSpeedBackward:=TRUE;
			T_Station_Work.TCtrlOnlineChange.xLockChange_S_WorkSpindleSpeed:=TRUE;
			IF (NOT(ptrTAxisZ^.T_CtrleSingle.xNotMoving) OR NOT(ptrTAxisZ^.T_CtrleSingle.xDone)) AND
	     		    NOT((ptrTAxisZ^.T_CtrleSingle.iFunction = 5) AND NOT(ptrTAxisZ^.T_CtrleSingle.xDone)) THEN
				ptrTAxisZ^.T_CtrleSingle.iFunction:=5;
				ptrTAxisZ^.T_CtrleSingle.xExecute:=TRUE;
			END_IF;
			IF NOT(ptrTAxisS^.T_CtrleSingle.xExecute) AND NOT(ptrTAxisS^.T_CtrleSingle.xNotMoving) THEN
				ptrTAxisS^.T_CtrleSingle.iFunction:=5;
				ptrTAxisS^.T_CtrleSingle.xExecute:=TRUE;
			END_IF;
			iStFct_Overload_StopProcess:=iStFct_Overload_StopProcess + 1;
			RETURN;
		2:	IF NOT(ptrTAxisZ^.T_CtrleSingle.xExecute) AND ptrTAxisZ^.T_CtrleSingle.xDone
			AND NOT(ptrTAxisS^.T_CtrleSingle.xExecute) AND ptrTAxisS^.T_CtrleSingle.xDone THEN
				T_Station_Work.THWWorkStation.TCtrlWork.xWorkingFinished:=TRUE;
				T_Station_Work.THWWorkStation.TCtrlWork.bPartQuality:=8;(* < Bearb. abgbr. > *)
				xStFct_HardwareError:=TRUE;
				IF xMaxTorqueActive THEN
					diStFct_TmpErrorNr:=16;		(* Wz Drehmoment Max überschritten *)
				ELSE
					diStFct_TmpErrorNr:=15;		(* Wz Drehmoment Überlast Aktiv *)
				END_IF;
			END_IF;
			RETURN;
		END_CASE;
	END_IF;
END_CASE;
END_ACTION
ACTION StationFunction_Ctrl_AxisBrake:
IF NOT(xAxisBrakeBlock) THEN
	IF NOT(ptrTAxisZ^.T_CtrleSingle.xPower) THEN
		IF NOT(ptrTCylBrakeReleaseZAxis^.T_CtrleCyl.T_Standard.xActivOff) AND NOT(ptrTCylBrakeReleaseZAxis^.T_CtrleCyl.xExecute) AND ptrTCylBrakeReleaseZAxis^.T_CtrleCyl.xDone THEN
			ptrTCylBrakeReleaseZAxis^.T_CtrleCyl.iFunction:=1;
			ptrTCylBrakeReleaseZAxis^.T_CtrleCyl.xExecute:=TRUE;
		END_IF;
	ELSE
		IF NOT(ptrTCylBrakeReleaseZAxis^.T_CtrleCyl.T_Standard.xActivOn) AND NOT(ptrTCylBrakeReleaseZAxis^.T_CtrleCyl.xExecute) AND ptrTCylBrakeReleaseZAxis^.T_CtrleCyl.xDone THEN
			ptrTCylBrakeReleaseZAxis^.T_CtrleCyl.iFunction:=2;
			ptrTCylBrakeReleaseZAxis^.T_CtrleCyl.xExecute:=TRUE;
		END_IF;
	END_IF;

END_IF;
END_ACTION
ACTION StationFunction_Ctrl_CalcProcWork:
(* Berechnung der Bearbeitungsarbeit *)
IF (iStFct_StepPrc = 3) THEN
	IF ptrTAxisZ^.T_CtrleSingle.xMovingForward AND NOT(ptrTAxisZ^.T_CtrleSingle.xNotMoving) THEN
		CASE T_ExchgParam.bToolSpindleActive OF
		1:	(* Maxon Spindel *)
			rTorqueForce:=T_Station_Parameter.T_TorqueSystem.rActual_Torque;		(* Maxon Spindel ist aktiv *)
		2:	(* Beckhoff Spindel L *)
			rTorqueForce:=T_Station_Parameter.T_TorqueSystem_L.rActual_Torque;		(* Beckhoff Spindel ist aktiv *)
		3:	(* Beckhoff Spindel M *)
			rTorqueForce:=T_Station_Parameter.T_TorqueSystem_M.rActual_Torque;		(* Beckhoff Spindel ist aktiv *)
		END_CASE;
		IF (rTorqueForce < 0.0) THEN
			rTorqueForce:=0.0;
		END_IF;
		IF NOT(xStFct_InitialCalcProcWork) THEN
			xStFct_InitialCalcProcWork:=TRUE;
			rStFct_ZSavePosition:=ptrTAxisZ^.T_LiveValue.lrActualPosition;
		END_IF;
		rStFct_ZCalcDistance:=rStFct_ZCalcDistance + (ptrTAxisZ^.T_LiveValue.lrActualPosition - rStFct_ZSavePosition);
		rStFct_ZSavePosition:=ptrTAxisZ^.T_LiveValue.lrActualPosition;
		diStFct_Counter:=diStFct_Counter + 1;
		rStFct_AddWorkForce:=(rStFct_AddWorkForce + rTorqueForce);
		rStFct_CalcWorkForce:=rStFct_AddWorkForce / DINT_TO_REAL(diStFct_Counter);
	END_IF;
ELSE
	xStFct_InitialCalcProcWork:=FALSE;
END_IF;
T_Station_Work.THWWorkStation.TCtrlWork.rProcessWork:=rStFct_CalcWorkForce * (rStFct_ZCalcDistance/1000.0);	(* Arbeit=Kraft(N)*Weg(m) *)
END_ACTION
ACTION StationFunction_Ctrl_CheckPos_Z:
xStFct_PositionOutRange_Z:=FALSE;
iStFct_PosErrorNr:=0;
IF (grZ_LoadPos > T_Station_Parameter.T_StProcess.rPositionEndMech) THEN
	iStFct_PosErrorNr:=27;	(* Z LadePos > Z Mech EndPos *)
ELSIF (grZ_WorkStartPos > T_Station_Parameter.T_StProcess.rPositionEndMech) THEN
	iStFct_PosErrorNr:=28;	(* Z Bearb StartPos > Z Mech EndPos *)
ELSIF (garPositionEndProcCalc[1] > T_Station_Parameter.T_StProcess.rPositionEndMech) THEN
	iStFct_PosErrorNr:=29;	(* Z Bearb EndPos > Z Mech EndPos *)
ELSIF (garCentringEndProcCalc[1] > T_Station_Parameter.T_StProcess.rPositionEndMech) THEN
	iStFct_PosErrorNr:=37;	(* Z ZentrierPos berechn. > Z Mech EndPos *)
ELSIF (T_Station_Parameter.T_StProcess.rZPositionCylindricalArea > T_Station_Parameter.T_StProcess.rPositionEndMech) THEN
	iStFct_PosErrorNr:=43;	(* Z WzZylinder Pos > Z Mech EndPos *)
ELSIF (T_Station_Parameter.T_StProcess.rPositionToolChange > T_Station_Parameter.T_StProcess.rPositionEndMech) THEN
	iStFct_PosErrorNr:=34;	(* Z WzWechsel Pos > Z Mech EndPos *)
ELSIF (grZ_LoadPos > grZ_WorkStartPos) AND
		(grZ_LoadPos > garPositionEndProcCalc[1]) THEN
	iStFct_PosErrorNr:=31;	(* Z LadePos: Stimmt nicht mit anderen Positionen überein *)
ELSIF (grZ_WorkStartPos < grZ_LoadPos) AND
		(grZ_WorkStartPos > garPositionEndProcCalc[1]) THEN
	iStFct_PosErrorNr:=32;	(* Z Bearb StartPos: Stimmt nicht mit anderen Positionen überein *)
ELSIF (garPositionEndProcCalc[1] < grZ_LoadPos) AND
		(garPositionEndProcCalc[1] < grZ_WorkStartPos) THEN
	iStFct_PosErrorNr:=33;	(* Z Bearb EndPos: Stimmt nicht mit anderen Positionen überein *)
END_IF;
IF (iStFct_PosErrorNr <> 0) THEN
	xStFct_PositionOutRange_Z:=TRUE;
END_IF;
END_ACTION
ACTION StationFunction_Ctrl_Controller_1:
(* Geschwindigkeitsregelung der Z1 Achse mittels der Kraftmessdose--> Konventioneller Regler *)
IF ptrTAxisZ^.T_CtrleSingle.xMovingForward THEN
	(* Konventionelle Regelung aber mit Override Funktion *)
	rStFct_V1:=	T_Station_Parameter.T_OnlineChange.rWorkingSpeedForward;
	rStFct_V2:=	T_Station_Parameter.T_OnlineChange.rWorkingSpeedForward/100.0;
	rStFct_S1:=	0.5;
	rStFct_S2:=	T_Station_Parameter.T_OnlineChange.rTorqueLevelHC;
	CASE T_ExchgParam.bToolSpindleActive OF
	1:	(* Maxon Spindel *)
		rStFct_M:=	T_Station_Parameter.T_TorqueSystem.rActual_Torque;		(* Maxon Spindel ist aktiv *)
	2:	(* Beckhoff Spindel L *)
		rStFct_M:=	T_Station_Parameter.T_TorqueSystem_L.rActual_Torque;	(* Beckhoff Spindel ist aktiv *)
	3:	(* Beckhoff Spindel M *)
		rStFct_M:=	T_Station_Parameter.T_TorqueSystem_M.rActual_Torque;	(* Beckhoff Spindel ist aktiv *)
	END_CASE;
	IF ((rStFct_S2 - rStFct_S1) <> 0.0) THEN
		rStFct_CalcZSpeed:=	rStFct_V1 -
							((rStFct_V1 - rStFct_V2) * ((rStFct_M - rStFct_S1)/(rStFct_S2 - rStFct_S1)));
	END_IF;
	IF ptrTSensorTorque^.T_CtrleCyl.xStatePosOff THEN
		IF (((rStFct_CalcZSpeed / rStFct_V1) *100.0) >= 0) THEN
			ptrTAxisZ^.T_CtrleSingle.dwOverride:=REAL_TO_DWORD((rStFct_CalcZSpeed / rStFct_V1) *100.0);
		ELSE
			ptrTAxisZ^.T_CtrleSingle.dwOverride:=1;
		END_IF;
	ELSE
		ptrTAxisZ^.T_CtrleSingle.dwOverride:=100;
	END_IF;
	IF (ptrTAxisZ^.T_CtrleSingle.dwOverride > 100) THEN
		ptrTAxisZ^.T_CtrleSingle.dwOverride:=100;
	ELSIF (ptrTAxisZ^.T_CtrleSingle.dwOverride < 1) THEN
		ptrTAxisZ^.T_CtrleSingle.dwOverride:=1;
	END_IF;
	ptrTAxisZ^.T_CtrleSingle.dwOverride:=REAL_TO_DWORD((DWORD_TO_REAL(ptrTAxisZ^.T_CtrleSingle.dwOverride)/100.0) * BYTE_TO_REAL(T_ExchgParam.byOverride));	(* Einstellung der Geschwindigkeit über das Poti *)
	IF (ptrTAxisZ^.T_CtrleSingle.dwOverride > 100) THEN
		ptrTAxisZ^.T_CtrleSingle.dwOverride:=100;
	ELSIF (ptrTAxisZ^.T_CtrleSingle.dwOverride < 1) THEN
		ptrTAxisZ^.T_CtrleSingle.dwOverride:=1;
	END_IF;
END_IF;
END_ACTION
ACTION StationFunction_Ctrl_Controller_2:
(* Geschwindigkeitsregelung der Z1 Achse mittels der Kraftmessdose--> Adaptive Vorschubssteuerung mit PID Regler für aufrecht erhaltene Drehmomentvorgabe *)
IF (iStFct_StepPrc = 3) THEN
	TONCalcTorque(IN:=TRUE,PT:=REAL_TO_TIME(INT_TO_REAL(T_Station_Parameter.T_StProcess.iZ_PID_FilterM)));
	diStepCount:=diStepCount + 1;
	rTorqueSpindleSensorSave:=rTorqueSpindleSensorSave + ptrTSensorTorque^.T_CtrleCyl.T_Analog.rPosIn;
	IF TONCalcTorque.Q THEN
		TONCalcTorque(IN:=FALSE);
		rTorqueSpindleSensor:=rTorqueSpindleSensorSave / DINT_TO_REAL(diStepCount);
		diStepCount:=0;
		rTorqueSpindleSensorSave:=0.0;
	END_IF;
	rOutMaxLimit:=(T_Station_Parameter.T_StProcess.rZ_PID_MaxSpeed/100.0) * BYTE_TO_REAL(T_ExchgParam.byOverride);	(* Einstellung der Geschwindigkeit über das Poti *)
	rOutMinLimit:=(T_Station_Parameter.T_StProcess.rZ_PID_MinSpeed/100.0) * BYTE_TO_REAL(T_ExchgParam.byOverride);		(* Einstellung der Geschwindigkeit über das Poti *)
	T_CtrlPara.rCtrlCycleTime:=0.001;
	T_CtrlPara.rKd:=T_Station_Parameter.T_StProcess.rZ_PID_Kd;
	T_CtrlPara.rKi:=T_Station_Parameter.T_StProcess.rZ_PID_Ki;
	T_CtrlPara.rKp:=T_Station_Parameter.T_StProcess.rZ_PID_Kp;
	T_CtrlPara.rOutMaxLimit:=rOutMaxLimit;
	T_CtrlPara.rOutMinLimit:=rOutMinLimit;
	FBPIDCTRL(	rSetpointValue:=T_Station_Parameter.T_StProcess.rZ_PID_Torque ,
						rActualValue:=rTorqueSpindleSensor ,
						T_CtrlPara:=T_CtrlPara);
	rStFct_CalcZSpeed:=FBPIDCTRL.rOut;
	T_Z_St1_Ctrle.diVelocityCommandValue:=LREAL_TO_DINT(rStFct_CalcZSpeed * -558349.25) ; (* 11166985 --> 20mm/s --> 1mm/s = 558349.25 *)
	RisingEdgeCountHC(CLK:=(ptrTAxisZ^.T_LiveValue.lrActualVelocity < 0));
	IF RisingEdgeCountHC.Q THEN
		wStFct_Status:=2;	(* 2 = < Wz Drehmom. HC> *)
		rStFct_SetZHCPosition:=ptrTAxisZ^.T_LiveValue.lrActualPosition;
		xStFct_CapturePosition:=TRUE;	(* Berechnung der Schnittgeschwindigkeit *)
		IF (rStFct_TmpDiffOverLimitPosition <> 0) THEN
			T_Station_Work.THWWorkStation.TCtrlWork.rDiffOverLimitPosition:=ptrTAxisZ^.T_LiveValue.lrActualPosition - T_Station_Work.THWWorkStation.TCtrlWork.rLastOverLimitPosition;
		END_IF;
		T_Station_Work.THWWorkStation.TCtrlWork.rLastOverLimitPosition:=ptrTAxisZ^.T_LiveValue.lrActualPosition;
		rStFct_TmpDiffOverLimitPosition:=T_Station_Work.THWWorkStation.TCtrlWork.rLastOverLimitPosition;
		T_Station_Work.THWWorkStation.TCtrlWork.iOverLimitCounterTorque:=T_Station_Work.THWWorkStation.TCtrlWork.iOverLimitCounterTorque + 1;
	END_IF;
ELSE
	diStepCount:=0;
	rTorqueSpindleSensorSave:=0.0;
	T_CtrlPara.xReset_I_Anteil:=TRUE;	(* Aufsummierter I-Anteil muss wieder zurückgesetzt werden, weil sonst dieser Wert mitgenommen wird *)
	FBPIDCTRL(	rSetpointValue:=T_Station_Parameter.T_StProcess.rZ_PID_Torque ,
				rActualValue:=rTorqueSpindleSensor ,
				T_CtrlPara:=T_CtrlPara);
	rTorqueSpindleSensor:=rTorqueSpindleSensorSave + ptrTSensorTorque^.T_CtrleCyl.T_Analog.rPosIn;
END_IF;
END_ACTION
ACTION StationFunction_Ctrl_Controller_3:
(* Geschwindigkeitsregelung der Z1 Achse mittels der Kraftmessdose--> Konventioneller Regler mit D Anteil und schnellerer Reaktionszeit so wie beim PID *)
IF (iStFct_StepPrc = 3) THEN
	TONCalcTorque(IN:=TRUE,PT:=REAL_TO_TIME(INT_TO_REAL(T_Station_Parameter.T_StProcess.iZ_D_FilterM)));
	diStepCount:=diStepCount + 1;
	rTorqueSpindleSensorSave:=rTorqueSpindleSensorSave + ptrTSensorTorque^.T_CtrleCyl.T_Analog.rPosIn;
	IF TONCalcTorque.Q THEN
		TONCalcTorque(IN:=FALSE);
		rTorqueSpindleSensor:=rTorqueSpindleSensorSave / DINT_TO_REAL(diStepCount);
		diStepCount:=0;
		rTorqueSpindleSensorSave:=0.0;
	END_IF;
	IF (T_Station_Parameter.T_StProcess.iWorkControlType = 3) THEN
		(* Konventionelle Regelung mit D-Regler mit Override Funktion *)
		rStFct_V1:=	(T_Station_Parameter.T_OnlineChange.rWorkingSpeedForward/100.0) * BYTE_TO_REAL(T_ExchgParam.byOverride);	(* Einstellung der Geschwindigkeit über das Poti *)
		rStFct_V2:=	T_Station_Parameter.T_OnlineChange.rWorkingSpeedForward/100.0;
		rStFct_S1:=	0.5;
		rStFct_S2:=	T_Station_Parameter.T_OnlineChange.rTorqueLevelHC;
		CASE T_ExchgParam.bToolSpindleActive OF
		1:	(* Maxon Spindel *)
			rStFct_M:=	T_Station_Parameter.T_TorqueSystem.rActual_Torque;		(* Maxon Spindel ist aktiv *)
		2:	(* Beckhoff Spindel L *)
			rStFct_M:=	T_Station_Parameter.T_TorqueSystem_L.rActual_Torque;	(* Beckhoff Spindel ist aktiv *)
		3:	(* Beckhoff Spindel M *)
			rStFct_M:=	T_Station_Parameter.T_TorqueSystem_M.rActual_Torque;	(* Beckhoff Spindel ist aktiv *)
		END_CASE;
		T_CtrlPara_D.rCtrlCycleTime:=0.001;
		T_CtrlPara_D.rKd:=T_Station_Parameter.T_StProcess.rZ_D_Kd;
		T_CtrlPara_D.rOutMaxLimit:=rStFct_V1;
		T_CtrlPara_D.rOutMinLimit:=rStFct_V2;
		rActualValue:=(rStFct_V1/rStFct_S2)*rTorqueSpindleSensor;		(* Drehmoment skalieren auf die Geschwindigkeit *)
		FBDCONTROL(	rActualValue:= rActualValue,
								T_CtrlPara:= T_CtrlPara_D);				
		
		IF ((rStFct_S2 - rStFct_S1) <> 0.0) THEN
			rStFct_CalcZSpeed_D:=	rStFct_V1 -
								((rStFct_V1 - rStFct_V2) * ((rStFct_M - rStFct_S1)/(rStFct_S2 - rStFct_S1)));
		END_IF;
		rStFct_CalcZSpeed:=rStFct_CalcZSpeed_D - FBDCONTROL.rOut;
		IF (rStFct_CalcZSpeed <= rStFct_V2) THEN
			rStFct_CalcZSpeed:=rStFct_V2;
		END_IF
		IF (rStFct_CalcZSpeed >= rStFct_V1) THEN
			rStFct_CalcZSpeed:=rStFct_V1;
		END_IF
		T_Z_St1_Ctrle.diVelocityCommandValue:=LREAL_TO_DINT(rStFct_CalcZSpeed * -558349.25) ;
	END_IF;
ELSE
	diStepCount:=0;
	rTorqueSpindleSensorSave:=0.0;
	rTorqueSpindleSensor:=rTorqueSpindleSensorSave + ptrTSensorTorque^.T_CtrleCyl.T_Analog.rPosIn;
END_IF;
END_ACTION
ACTION StationFunction_Ctrl_Controller_O:
(* Zweipunkte Regler der O Achse mittels der Kraftmessdose--> Hier wird nur ein oder ausgeschaltet der O Achse *)
IF ptrTAxisZ^.T_CtrleSingle.xMovingForward AND (T_Station_Parameter.T_StProcess.rO_Ctrl_HystereseOffset <> 0) AND (T_Station_Parameter.T_StProcess.rWorkingSpeedOscillation > 0.0) THEN
	IF ptrTSensorTorque^.T_CtrleCyl.xStatePosOff THEN
		IF (T_Station_Work.THWWorkStation.TCtrlWork.iProgressBar_Torque > T_Station_Parameter.T_StProcess.rO_Ctrl_TorquePercent_OFF) AND QxFastStrokeOn_St1 AND NOT(xBlockActivateOAxis) THEN
			QxFastStrokeOn_St1:=FALSE;		(* Schwellwert überschritten und deshalb muss ausgeschaltet werden *)
			xBlockActivateOAxis:=TRUE;
		ELSE
			IF (T_Station_Parameter.T_StProcess.rO_Ctrl_HystereseOffset > 0) THEN
				(* Hystere ist Positiv eingestellt und deshalb muss das Drehmoment um diesen Hysteresoffset steigen damit der Schnellhub wieder eingeschaltet wird *)
				IF (T_Station_Work.THWWorkStation.TCtrlWork.iProgressBar_Torque > (T_Station_Parameter.T_StProcess.rO_Ctrl_TorquePercent_OFF + T_Station_Parameter.T_StProcess.rO_Ctrl_HystereseOffset)) THEN
					QxFastStrokeOn_St1:=TRUE;		(* Schnellhub kann wieder eingeschaltet werden *)
				END_IF;
				IF (T_Station_Work.THWWorkStation.TCtrlWork.iProgressBar_Torque < T_Station_Parameter.T_StProcess.rO_Ctrl_TorquePercent_OFF) THEN
					(* Bei positiver Hysteres muss es zuerst wieder den Schwellwert unterschreiten bis es wider freigeben kann um es dann wieder zu deaktivierren *)
					xBlockActivateOAxis:=FALSE;
				END_IF;
			ELSE
				(* Hystere ist Negativ eingestellt und deshalb muss das Drehmoment um diesen Hysteresoffset sinken damit der Schnellhub wieder eingeschaltet wird *)
				IF (T_Station_Work.THWWorkStation.TCtrlWork.iProgressBar_Torque < (T_Station_Parameter.T_StProcess.rO_Ctrl_TorquePercent_OFF - ABS(T_Station_Parameter.T_StProcess.rO_Ctrl_HystereseOffset))) THEN
					QxFastStrokeOn_St1:=TRUE;		(* Schnellhub kann wieder eingeschaltet werden *)
					xBlockActivateOAxis:=FALSE;
				END_IF;
			END_IF;
		END_IF;
	END_IF;
ELSE
	xBlockActivateOAxis:=FALSE;
END_IF;
END_ACTION
ACTION StationFunction_Ctrl_Controller_S:
(* Drehzahlregler der S Achse  mittels der Kraftmessdose--> Konventioneller Regler aber ohne Override da das Override nicht grösser werden darf als 100
   Den Min Max Wert kann man hier auch als Max definieren, d.h. bei ansteigendem Drehmoment wird die Drehzahl höher und deshalb funktioniert das Override nicht *)
IF ptrTAxisZ^.T_CtrleSingle.xMovingForward AND (T_Station_Parameter.T_StProcess.rWorkingSpindleSpeedMinMax <> 0.0) THEN
	(* Konventionelle Regelung aber ohne Override Funktion *)
	rStFct_V1:=	T_Station_Parameter.T_OnlineChange.rWorkingSpindleSpeed;
	rStFct_V2:=	T_Station_Parameter.T_StProcess.rWorkingSpindleSpeedMinMax;
	rStFct_S1:=	0.5;
	rStFct_S2:=	T_Station_Parameter.T_OnlineChange.rTorqueLevelHC;
	CASE T_ExchgParam.bToolSpindleActive OF
	1:	(* Maxon Spindel *)
		rStFct_M:=	T_Station_Parameter.T_TorqueSystem.rActual_Torque;		(* Maxon Spindel ist aktiv *)
	2:	(* Beckhoff Spindel L *)
		rStFct_M:=	T_Station_Parameter.T_TorqueSystem_L.rActual_Torque;	(* Beckhoff Spindel ist aktiv *)
	3:	(* Beckhoff Spindel M *)
		rStFct_M:=	T_Station_Parameter.T_TorqueSystem_M.rActual_Torque;	(* Beckhoff Spindel ist aktiv *)
	END_CASE;
	IF ((rStFct_S2 - rStFct_S1) <> 0.0) THEN
		rStFct_CalcZSpeed:=	rStFct_V1 -
							((rStFct_V1 - rStFct_V2) * ((rStFct_M - rStFct_S1)/(rStFct_S2 - rStFct_S1)));
	END_IF;
	IF (rStFct_CalcZSpeed > 0) THEN
		IF ptrTSensorTorque^.T_CtrleCyl.xStatePosOff THEN
			IF (ABS(lrSaveSSpeed - rStFct_CalcZSpeed) > 20) THEN	(* Geschwindigkeitsübergabe nur wenn Änderung grösser ist als 20min-1 *)
				IF NOT(ptrTAxisS^.T_CtrleSingle.xExecute) AND ptrTAxisS^.T_CtrleSingle.xDone AND
				     NOT(ptrTAxisS^.T_CtrleSingle.xErr) AND NOT(ptrTAxisS^.T_CtrleSingle.xNotMoving) THEN
					xSetDefaultSpeedS:=FALSE;
					lrSaveSSpeed:=rStFct_CalcZSpeed;
					ptrTAxisS^.T_CtrleSingle.iFunction:=12;
					ptrTAxisS^.T_CtrleSingle.lrVelocity:=rStFct_CalcZSpeed;
					ptrTAxisS^.T_CtrleSingle.xExecute:=TRUE;
				END_IF;
			END_IF;
		ELSE
			IF NOT(xSetDefaultSpeedS) THEN
				IF NOT(ptrTAxisS^.T_CtrleSingle.xExecute) AND ptrTAxisS^.T_CtrleSingle.xDone AND
				     NOT(ptrTAxisS^.T_CtrleSingle.xErr) AND NOT(ptrTAxisS^.T_CtrleSingle.xNotMoving) THEN
					xSetDefaultSpeedS:=TRUE;
					ptrTAxisS^.T_CtrleSingle.iFunction:=12;
					ptrTAxisS^.T_CtrleSingle.lrVelocity:=T_Station_Parameter.T_OnlineChange.rWorkingSpindleSpeed;
					ptrTAxisS^.T_CtrleSingle.xExecute:=TRUE;
				END_IF;
			END_IF;
		END_IF;
	END_IF;
ELSE
	xSetDefaultSpeedS:=FALSE;
END_IF;
END_ACTION
ACTION StationFunction_Ctrl_End:
IF xStFct_SetEnd THEN
	xStFct_End:=TRUE;
	xStFct_InitStep:=FALSE;
	xStFct_SetEnd:=FALSE;
	xStFct_Stop:=FALSE;
	xStFct_StartMainPrc:=FALSE;
	xStFct_InitMainCtr:=FALSE;
	xStFct_StartMainCtr:=FALSE;
	xStFct_Start:=FALSE;
	xStFct_HardwareError:=FALSE;
	xStFct_QuitErr:=FALSE;
	xStFct_Error:=FALSE;
	diStFct_ErrorNr:=0;
	xStFct_InitError:=FALSE;
	xStFct_Freeze:=FALSE;
	xStFct_Abord:=FALSE;
	xStFct_Reset:=FALSE;
	xStFct_StartPrc_Parallel:=FALSE;
	iStFct_StepPrc_Parallel:=1;
	xStFct_InitStep_Parallel:=FALSE;
	xStFct_ToolDeflectionActiveStopProcess:=FALSE;
	xStFct_ToolClampInactiveStopProcess:=FALSE;
	T_Station_Work.TCtrlOnlineChange.xLockChange_S_WorkSpindleSpeed:=TRUE;
	xStFct_DeflCalibError:=FALSE;
	xStFct_TorqueCalibError:=FALSE;
	xStFct_InitStopProcess:=FALSE;
	IF (iStationFunctionNr = 4) OR (iStationFunctionNr = 5) THEN
		T_Station_Work.THWWorkStation.TCtrlWork.xWorkingFinished:=FALSE;
	END_IF;
	IF xSecurityCircuitOn THEN
		T_Station_Work.TCtrlOnlineChange.xLockChangeCylToolDeflectionForce:=FALSE;
		T_Station_Work.TCtrlOnlineChange.xLockChangeCylToolTorqueLevel:=FALSE;
	END_IF;
	T_Station_Work.THWWorkStation.TCtrlWork.xSparkOutActive:=FALSE;
	gxWP_Analyse_ActiveWork:=FALSE;
	gxWP_Analyse_ActiveInfeed:=FALSE;
	gxWP_Analyse_ActiveCentering:=FALSE;
	IF xStFct_TmpSaveOffset THEN
		(* Im Fehlerfall oder die Funktion gestoppt wird muss der alte Wert wieder übergeben werden *)
		xStFct_TmpSaveOffset:=FALSE;
		IF T_Station_Work.THWWorkStation.TCtrlWork.xActiveCalibrateToolDeflection THEN
			T_Station_Parameter.T_Fct_SpindleCalibration.arOffsetToolDeflection[1]:=rStFct_TmpOffsetDeflection;
		END_IF;
		IF T_Station_Work.THWWorkStation.TCtrlWork.xActiveCalibrateToolTorque THEN
			T_Station_Parameter.T_Fct_SpindleCalibration.arOffsetToolTorque[1]:=rStFct_TmpOffsetTorque;
		END_IF;
		IF xSafetyCircuitOn THEN
			(* Zylinder für Auslenkung-->mit Workauslenkkraft *)
			IF ptrTCylToolDeflection^.T_CtrleCyl.xDone THEN
				ptrTCylToolDeflection^.T_CtrleCyl.iFunction:=2;
				ptrTCylToolDeflection^.T_Config.tDelayOn:=T#0s;
				ptrTCylToolDeflection^.T_CtrleCyl.T_Analog.rForceIn:=T_Station_Parameter.T_OnlineChange.rForceDeflection;
				ptrTCylToolDeflection^.T_CtrleCyl.xExecute:=TRUE;
			END_IF;
		END_IF;
	END_IF;
	xBlockCheckLimitSwitch:=FALSE;
	xBlockSetFastVelZAxis:=FALSE;
END_IF;
END_ACTION
ACTION StationFunction_Ctrl_Error:
xStFct_ErrorActuator:=	ptrTAxisZ^.T_CtrleSingle.xErr OR ptrTAxisS^.T_CtrleSingle.xErr;
xStFct_ExecuteActuator:=	NOT(ptrTAxisZ^.T_CtrleSingle.xExecute) AND NOT(ptrTAxisS^.T_CtrleSingle.xExecute);

